FUNCTION_BLOCK FB_CommandWithStruct EXTENDS CommandBase
VAR
	{attribute 'PlcCommandInput'}
	stInputArgs		: ST_CommandArgs;
	{attribute 'PlcCommandInput'}
	nNumber			: INT;
	{attribute 'PlcCommandInput'}
	eEnum			: E_EnumType;
	
	{attribute 'PlcCommandOutput'}
	stOutputArgs	: ST_CommandArgs;
	{attribute 'PlcCommandOutput'}
	fFloat			: REAL;
END_VAR

SUPER^();

// Will be called when ``stHandshake.bExecute`` changes to ``true`` one cycle and in the same cycle.
METHOD PROTECTED Init
stOutputArgs := stInputArgs;
fFloat := stInputArgs.fFloat;
Finish(E_CommandResultCode.Done);
END_METHOD

END_FUNCTION_BLOCK

(* stored: Version 1.1.0.1, ProductVersion 3.1.4022.12
   POU FB_CommandWithStruct: Id {21088bbb-8d5b-0fc1-300f-5438a5c6f591}, SpecialFunc None
   Method Init: Id {3f7dc758-bb49-04b9-3246-0edbe2c710b8} *)
